PROGRAM PRG_Example
VAR_INPUT
    bStart : BOOL;
END_VAR
VAR_OUTPUT
    bRunning : BOOL;
END_VAR
VAR
    nCycleCount : DINT;
END_VAR

IF bStart THEN
    bRunning := TRUE;
    nCycleCount := nCycleCount + 1;
END_IF;

END_PROGRAM

(* stored: Version 1.1.0.1
   POU PRG_Example: Id {11111111-1111-1111-1111-111111111111}, SpecialFunc None *)
